TYPE "tAutoConveyor"
VERSION : 0.8
   STRUCT
      "standard" : "tAutoStandard";
   END_STRUCT;

END_TYPE
